Fanuc KAREL source: kt00050.KL

-- PROVISIONAL review KL for V1013-1; original PC SHA256 b995118ed8888c147090bc16c8f1454170cfb5d5161cc5721ee08faa5348b7e3
-- Incomplete behavior may be omitted. Consult companion uncertainty JSON. Do not deploy.
PROGRAM KT00050
%NOLOCKGROUP
VAR
  I2 : INTEGER
  OUT : REAL
-- UNRESOLVED_DECL Y1 type=002018
BEGIN
  -- UNRESOLVED_PC offsets 5-19; opcodes 2E,22,9D,33,B2
  -- UNRESOLVED_PC offsets 24-35; opcodes 2E,23
  -- UNRESOLVED_PC offsets 40-63; opcodes 22,9D,33,B1,21,53,64,23
  -- UNRESOLVED_PC offsets 68-72; opcodes 7F
END KT00050
